// Mitsubishi GX Works2 project: fk3n_test_in_out   PLC: FX3U/FX3UC

PROGRAM MAIN
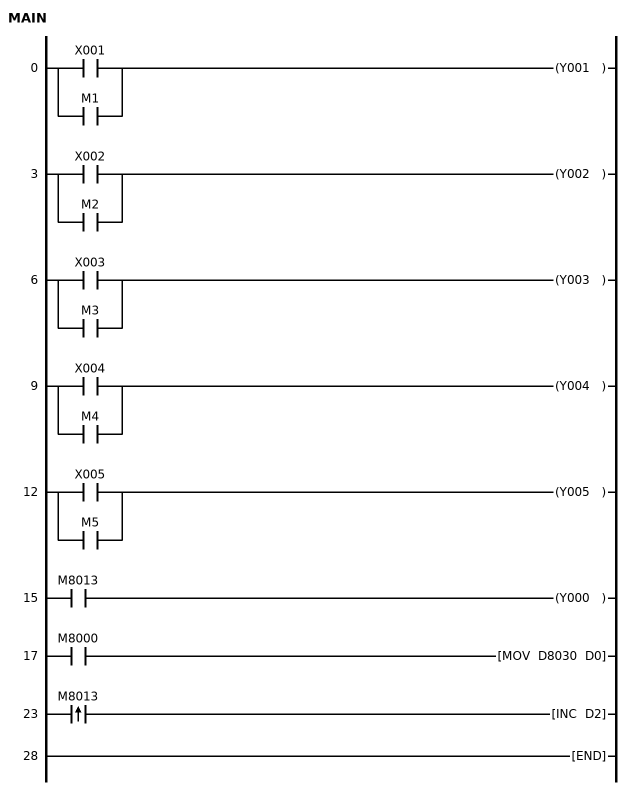
0     LD      X001
      OR      M1
      OUT     Y001
3     LD      X002
      OR      M2
      OUT     Y002
6     LD      X003
      OR      M3
      OUT     Y003
9     LD      X004
      OR      M4
      OUT     Y004
12    LD      X005
      OR      M5
      OUT     Y005
15    LD      M8013
      OUT     Y000
17    LD      M8000
      MOV     D8030 D0
23    LDP     M8013
      INC     D2
28    END
END_PROGRAM
